(*

.. <legal notes>

legal notes
=================
| SPDX-FileCopyrightText: © 2026 Oleksandr Tiutyk <trofimich@gmail.com>
| SPDX-License-Identifier: LGPL-3.0-only
| For details check: LGPL-3.0-only_

.. _LGPL-3.0-only: https://www.gnu.org/licenses/lgpl-3.0.en.html

.. </legal notes>

*)

FUNCTION_BLOCK TestAutomationRunner EXTENDS TOF_AutomationEngine.AutomationRunner<1>
VAR
	_ClassName : STRING := __POUNAME();

	_TestAutomationUnit : TestAutomationController;
	
	_AutomationControllers : ARRAY [0.._ControllerCount - 1] OF TOF_AutomationEngine.IAutomationController := [_TestAutomationUnit];
END_VAR

{attribute 'monitoring' := 'call'}
PROPERTY ClassName : STRING
GET
ClassName := _ClassName;
END_GET
END_PROPERTY

{attribute 'monitoring' := 'call'}
PROPERTY Controllers : REFERENCE TO ARRAY [0.._ControllerCount - 1] OF TOF_AutomationEngine.IAutomationController
GET
Controllers REF= _AutomationControllers;
END_GET
END_PROPERTY

{attribute 'monitoring' := 'call'}
PROPERTY NamespaceName : STRING
GET
NamespaceName := CurrentNamespace.Name;
END_GET
END_PROPERTY

{attribute 'monitoring' := 'call'}
PROPERTY SelfSize : ULINT
GET
SelfSize := XSIZEOF(THIS^);
END_GET
END_PROPERTY

END_FUNCTION_BLOCK

(* stored: Version 1.1.0.1, ProductVersion 3.1.4026.17
   POU TestAutomationRunner: Id {c1247552-9649-4dd8-ba25-e7403c6b5f57}, SpecialFunc None
   Property ClassName: Id {5636aa4d-d259-43df-a593-998a4fd52855}
   Get Get: Id {c7dfc2e6-64b3-405f-a918-1b3330edf922}
   Property Controllers: Id {39c079df-61e9-4be3-9044-7d9478bda0d8}
   Get Get: Id {c09259b0-9665-4cf9-b334-c96212dd0ff4}
   Property NamespaceName: Id {a18d2e63-2e16-4e45-b147-be3c7679499c}
   Get Get: Id {11210dc0-58af-4402-9e9b-c1c9861a5ae8}
   Property SelfSize: Id {7ce44a07-5152-4f85-ae69-7ca40274ffdc}
   Get Get: Id {fd68cde4-92c0-487c-99ce-cd65d169fd6e} *)
